(* PLC project Tc2_Utilities.DEC_TO_BCD Demo, tc3-libraries-kb TwinCAT 3.1 *)
(* stored: creationDateTime 2026-05-11T00:00:00, modificationDateTime 2026-05-11T00:00:00 *)

PROGRAM P_Demo_DEC_TO_BCD
  VAR
    fbDEC_TO_BCD : DEC_TO_BCD;  (* DEC_TO_BCD 实例 *)
    decValue : BYTE := 47;  (* PLC 内部十进制值 *)
    bcdOutput : BYTE;  (* 送往 7 段译码模块的 BCD 字节 *)
  END_VAR

// =============================================================================
// 场景：把工位号 0..99 编码为 BCD 字节，输出到老式 7 段显示模块。
// 价值：封装位运算，意图清晰。
// 验证：改 decValue := 47，观察 bcdOutput 应为 16#47；改 99 应为 16#99；改 100 应为 16#60（脱离合法 BCD）。
// 验证步骤：
//   1. 右键 PLC 项目 → Import PLCopenXML → 选本文件
//   2. 引用 Tc2_Utilities（References → Add library）
//   3. 编译 → 登录 → 运行；按上方『验证』行的指示在线写值观察
// =============================================================================

decValue := LIMIT(0, decValue, 99);  // 工程保护：超范围会得到非法 BCD
fbDEC_TO_BCD(DECIN := decValue, BCDOUT => bcdOutput);
END_PROGRAM
